# EPICS substitutions: ek9000App/Db/EL3204.substitutions
file EL3204.template
{ 	pattern
	{
		TERMINAL,

	}
	{
	}
}

	}
	{
	}
}

	}
	{
	}
}

	}
	{
	}
}
